TYPE ST_MotorErrors :
STRUCT	
	Thermal					: BOOL;
	Maintenance				: BOOL;
END_STRUCT
END_TYPE

(* stored: Version 1.1.0.1, ProductVersion 3.1.4020.12
   DUT ST_MotorErrors: Id {222023a1-ca92-401f-a8ee-c723edd69744} *)
